// TIA Portal V17 export
// export: Created 2025-03-07T09:24:33.0643277Z, ExportSetting WithDefaults, DisplayName Totally Integrated Automation Portal, DisplayVersion V17 Update 8, DisplayName TIA Portal Openness, DisplayVersion V17 Update 8, DisplayName TIA Portal Version Control Interface, DisplayVersion V17, DisplayName SINAMICS Startdrive Advanced, DisplayVersion V17 SP2, DisplayName SINAMICS Startdrive G110M, G120, G120C, G120D, G120P, G115D, DisplayVersion V17 SP2, DisplayName SINAMICS Startdrive G130, G150, S120, S150, SINAMICS MV, S210, DisplayVersion V17 SP2, DisplayName STEP 7 Professional, DisplayVersion V17 Update 8, DisplayName SINUMERIK ONE STEP 7 Toolbox, DisplayVersion V17 Update 12, DisplayName SINUMERIK 840D sl STEP 7 Toolbox, DisplayVersion V17 Update 12, DisplayName STEP 7 Safety, DisplayVersion V17 Update 6, DisplayName WinCC Advanced, DisplayVersion V17 Update 8
VAR_GLOBAL   // PLC tag table "TAGS_SAFETY_IO_PROGRAM"
   FEEDBACK_OFF_E_STOP_IN AT %I143.1 : Bool;   // FEEDBACK OFF E-STOP INPUT
   FEEDBACK_OFF_E_STOP_RST_STR_IN AT %I143.2 : Bool;   // FEEDBACK OFF E-STOP RESET START INPUT
   FEEDBACK_OFF_MACHINE_E_STOP_IN AT %M10030.2 : Bool;   // FEEDBACK OFF MACHINE E-STOP INPUT
   FEEDBACK_OFF_MACHINE_E_STOP_RST_STR_IN AT %M10030.3 : Bool;   // FEEDBACK OFF MACHINE E-STOP RESET START INPUT
   SAFE_INPUT_MACH_E_STOP AT %I300.0 : Bool;   // SAFETY INPUT MACHINE EMERGENCY STOP
   SAFE_OUT_E_STOP_OK AT %Q330.0 : Bool;   // SAFETY OUTPUT EMERGENCY STOP OK
   SAFE_OUT_MACHINE_E_STOP_OK AT %M10050.1 : Bool;   // SAFETY OUTPUT EMERGENCY STOP OK
END_VAR
